// TIA Portal V21 export
VAR_GLOBAL   // PLC tag table "K_Stazioni"
END_VAR
VAR_GLOBAL CONSTANT   // user constants
   K_Stazione_PompaAcidificazioneVascaEvaporati : Int := 1;
   K_Stazione_Acidificazione1 : Int := 2;
   K_Stazione_Acidificazione2 : Int := 3;
   K_Stazione_Acidificazione3 : Int := 4;
   K_Stazione_Acidificazione4 : Int := 5;
   K_Stazione_BermaProntoFresco : Int := 6;
   K_Stazione_BermaPomodoro : Int := 7;
   K_Stazione_Cernita1 : Int := 8;
   K_Stazione_CFT_MVRAEstrazione1 : Int := 9;
   K_Stazione_CFT_MVRAEstrazione2 : Int := 10;
   K_Stazione_CFT_MVRBEstrazione1 : Int := 11;
   K_Stazione_CFT_MVRBFinitore1 : Int := 12;
   K_Stazione_CFT_MVRBFinitore2 : Int := 13;
   K_Stazione_CocleaIFT1_2 : Int := 14;
   K_Stazione_D1 : Int := 15;
   K_Stazione_D2 : Int := 16;
   K_Stazione_Decanter1 : Int := 17;
   K_Stazione_Decanter2 : Int := 18;
   K_Stazione_Decanter3 : Int := 19;
   K_Stazione_Ghizzoni : Int := 20;
   K_Stazione_IFT3 : Int := 21;
   K_Stazione_IFT5 : Int := 22;
   K_Stazione_IFT6 : Int := 23;
   K_Stazione_Lince1 : Int := 24;
   K_Stazione_Lince2 : Int := 25;
   K_Stazione_Lince3 : Int := 26;
   K_Stazione_Lince4 : Int := 27;
   K_Stazione_PICO1 : Int := 28;
   K_Stazione_PICO2 : Int := 29;
   K_Stazione_PompaAlimentazioneDecanter : Int := 30;
   K_Stazione_PompaAlimentazioneHB1 : Int := 31;
   K_Stazione_PompaAlimentazioneHB1_HB2 : Int := 32;
   K_Stazione_PompaAlimentazioneHB2 : Int := 33;
   K_Stazione_PompaAlimentazioneHB3 : Int := 34;
   K_Stazione_PompaInvio1 : Int := 35;
   K_Stazione_PompaCrema1 : Int := 36;
   K_Stazione_PompaConcentrato1 : Int := 37;
   K_Stazione_PompaInvio2 : Int := 38;
   K_Stazione_PompaCrema2 : Int := 39;
   K_Stazione_PompaInvio3 : Int := 40;
   K_Stazione_PompaCrema3 : Int := 41;
   K_Stazione_PompaInvio4 : Int := 42;
   K_Stazione_PompaCrema4 : Int := 43;
   K_Stazione_PompaInvio5 : Int := 44;
   K_Stazione_PompaCrema5 : Int := 45;
   K_Stazione_PompaInvio6 : Int := 46;
   K_Stazione_PompaInvio7 : Int := 47;
   "K_Stazione_PompaNastroIFT1-2" : Int := 48;
   K_Stazione_PompaRecuperoIFT1 : Int := 49;
   K_Stazione_PompaRecuperoIFT2 : Int := 50;
   K_Stazione_PompaRecuperoPizza : Int := 51;
   K_Stazione_Salsina1 : Int := 52;
   K_Stazione_Salsina2 : Int := 53;
   K_Stazione_Salsina3 : Int := 54;
   K_Stazione_Salsina4 : Int := 55;
   K_Stazione_Scrambler : Int := 56;
   K_Stazione_TorchioScrambler : Int := 57;
   K_Stazione_Separapelli1Sx : Int := 58;
   K_Stazione_Separapelli2Dx : Int := 59;
   K_Stazione_Serpentino : Int := 60;
   K_Stazione_SgrondatoreP54 : Int := 61;
   K_Stazione_TorchioSgrondatoreP54 : Int := 62;
   K_Stazione_SgrondatoreP55 : Int := 63;
   "K_Stazione_T150_1/2EffettoP05" : Int := 64;
   "K_Stazione_T150_1/2EffettoP07" : Int := 65;
   K_Stazione_T150_3EffettofinitoreP02 : Int := 66;
   K_Stazione_TrituratoD1 : Int := 67;
   K_Stazione_TrituratoD2 : Int := 68;
   K_Stazione_TrituratoBrovatrice : Int := 69;
   K_Stazione_Vasca30Quintali : Int := 70;
   K_Stazione_VascaDecanter : Int := 71;
   K_Stazione_VascaEvaporatiP134 : Int := 72;
   K_Stazione_VascaEvaporatiP135 : Int := 73;
   K_Stazione_VascaMix : Int := 74;
   K_Stazione_VascaPolpa1 : Int := 75;
   K_Stazione_VascaPolpa2 : Int := 76;
   K_Stazione_VascaEvaporati : Int := 77;
   K_Stazione_CatelliLogicon : Int := 78;
   K_Stazione_CFT10t : Int := 79;
   K_Stazione_CatelliOhmico : Int := 80;
   K_Stazione_Goglio : Int := 81;
   K_stazione_CatelliConcentrato : Int := 82;
   K_Stazione_PastorizzatoreGoglio2 : Int := 83;
   K_Stazione_VascaSemiconcentrato : Int := 84;
   K_Stazione_FBR200Kg : Int := 85;
   K_Stazione_IFT1 : Int := 86;
   K_Stazione_IFT2 : Int := 87;
   K_Stazione_VascaCrema : Int := 88;
   K_Stazione_HB1 : Int := 89;
   K_Stazione_HB2 : Int := 90;
   K_Stazione_HB3 : Int := 91;
   K_Stazione_FMCPolpa : Int := 92;
   K_Stazione_IFT4 : Int := 93;
   K_Stazione_CircolazioneCrema : Int := 94;
   K_Stazione_Scottatrice : Int := 95;
   K_Stazione_LineaIFT_A : Int := 96;
   K_Stazione_LineaIFT_B : Int := 97;
   K_Stazione_LineaIFT_C : Int := 98;
   K_Stazione_LineaIFT_D : Int := 99;
END_VAR
